{attribute 'linkalways'} 
{attribute 'no_explicit_call' := 'This FB is a CLASS and must be accessed using methods or properties'}
{attribute 'enable_dynamic_creation'}
FUNCTION_BLOCK _ETcVnPrototypeClusterer EXTENDS EnumDatatypeBase
VAR
	localData : ETcVnPrototypeClusterer;
	activeData : REFERENCE TO ETcVnPrototypeClusterer;
	enumBaseDatatype : _UDINT(localData);
END_VAR

METHOD PRIVATE AddLocalEnumeration
VAR_INPUT
	Enumeration : T_MAXSTRING;
	Value : ETcVnPrototypeClusterer;
END_VAR
AddEnumeration(Enumeration, Value);
END_METHOD

PROPERTY PUBLIC Address : PVOID
GET
Address := ADR(activeData);
END_GET
END_PROPERTY

METHOD PUBLIC ClearReference
VAR_INPUT
END_VAR
activeData REF= localData;
SetBaseDatatypeReference();
END_METHOD

METHOD PUBLIC Clone : I_Datatype
VAR
    pClone : POINTER TO _ETcVnPrototypeClusterer;
END_VAR
pClone := __NEW(_ETcVnPrototypeClusterer(InitialValue := Value));
Clone := pClone^;
END_METHOD

METHOD FB_init : BOOL
VAR_INPUT
	bInitRetains : BOOL; // if TRUE, the retain variables are initialized (warm start / cold start)
	bInCopyCode : BOOL;  // if TRUE, the instance afterwards gets moved into the copy code (online change)
	InitialValue : ETcVnPrototypeClusterer;
END_VAR
localData := InitialValue;
AddBaseDatatype(enumBaseDatatype);
ClearReference();

AddLocalEnumeration('TCVN_PC_NOVELTY_DETECTOR', ETcVnPrototypeClusterer.TCVN_PC_NOVELTY_DETECTOR);
AddLocalEnumeration('TCVN_PC_CLUSTERER', ETcVnPrototypeClusterer.TCVN_PC_CLUSTERER);
END_METHOD

PROPERTY PUBLIC Identifier : T_MAXSTRING
GET
Identifier := 'ETcVnPrototypeClusterer';
END_GET
END_PROPERTY

METHOD IsEnumeratorValueEqual : BOOL
VAR_INPUT
	Enumerator : I_KeyValueForwardEnumerator;
END_VAR
VAR
	storedValue : ETcVnPrototypeClusterer;
END_VAR
IF NOT Enumerator.TryGet(storedValue) THEN
	RETURN;
END_IF

IsEnumeratorValueEqual := storedValue = activeData;
END_METHOD

METHOD PUBLIC MakeReferenceTo
VAR_INPUT
	ReferenceTarget : REFERENCE TO ETcVnPrototypeClusterer;
END_VAR
activeData REF= ReferenceTarget;
SetBaseDatatypeReference();
END_METHOD

METHOD PROTECTED SetBaseDatatypeReference
VAR_INPUT
END_VAR
enumBaseDatatype.MakeReferenceTo(activeData);
END_METHOD

PROPERTY PUBLIC Size : UDINT
GET
Size := SIZEOF(activeData);
END_GET
END_PROPERTY

METHOD TryMakeReferenceTo : BOOL
VAR_INPUT
	Target : I_Datatype;
END_VAR
VAR
	targetAsEnum : I_EnumDatatype;
	pTargetData : POINTER TO ETcVnPrototypeClusterer;
END_VAR
IF NOT Target.TryResolveAsEnumDatatype(targetAsEnum) THEN
	RETURN;
END_IF

IF targetAsEnum.Identifier <> Identifier THEN
	RETURN;
END_IF

pTargetData := Target.Address;
activeData REF= pTargetData^;
SetBaseDatatypeReference();
TryMakeReferenceTo := TRUE;
END_METHOD

PROPERTY PUBLIC Value : ETcVnPrototypeClusterer
GET
Value := activeData;
END_GET
SET
activeData := Value;
END_SET
END_PROPERTY

END_FUNCTION_BLOCK

(* stored: Version 1.1.0.1, ProductVersion 3.1.4024.12
   POU _ETcVnPrototypeClusterer: Id {89865f35-a855-4d84-b139-ff6c1019d7f7}, SpecialFunc None
   Folder Constructor: Id {4d849d09-b42c-4612-b751-9754bd6127fc}
   Folder Private: Id {a15ca895-ab8b-469d-bd2d-c915e5c9c382}
   Folder Protected: Id {6aebfd5f-71a5-4ad9-b65c-0177d12b4608}
   Method AddLocalEnumeration: Id {a4ae2f54-1c3c-4038-ab38-c1b378479abc}
   Property Address: Id {467cd426-e7f0-4851-88eb-b8398657c6a3}
   Get Get: Id {089f2cd8-502d-4392-b709-33417907b773}
   Method ClearReference: Id {89cee03a-ce65-47ea-955d-3799a487583d}
   Method Clone: Id {5b514904-5d0d-4a8c-81a6-c46af0c4d27b}
   Method FB_init: Id {27cb1c6d-491c-4d0a-a088-0264899651c9}
   Property Identifier: Id {bc633fe0-7d42-4c0a-9ec2-dadb8b23ba40}
   Get Get: Id {f6b6ddf5-43a0-467c-a567-e21f9ee218b4}
   Method IsEnumeratorValueEqual: Id {176b7f3c-9cb4-4784-8a56-f6e287ba82a0}
   Method MakeReferenceTo: Id {b035f1f7-e8cd-4b8b-b76c-4d37f49cb3fd}
   Method SetBaseDatatypeReference: Id {2d8a11a2-55fa-4711-b19c-044d22457e81}
   Property Size: Id {cd53300a-c5c8-4dc7-911a-167c8150e8e4}
   Get Get: Id {a018cf64-a7da-470a-8527-b8cba13fc873}
   Method TryMakeReferenceTo: Id {a8b8fb8f-1573-4316-b77c-41cfdeeb2c38}
   Property Value: Id {a0055dd9-b759-4e47-82ae-f20efece2a7f}
   Get Get: Id {75a33ebc-5dca-44d0-b770-fb87661ff934}
   Set Set: Id {ad40d8c3-3a78-434d-a5e5-0d3323f18467} *)
